# EPICS StreamDevice protocol: gemorcSup/devgemorc.proto
OutTerminator = CR;
InTerminator = CR;

getID {
	out "id";
	in "%#s";
}

initialise {
	out "in";
	in "OK";
}

re_zero_to_datum {
	out "da";
	in "OK";
}

stopNextInit {
	out "si";
	in "OK";
}

start {
	out "st";
	in "OK";
}

stop {
	out "sp";
	in "OK";
}

setWidth {
	out "ww%03d";
	in "OK";
	@init {out "rq"; in "%*16c%03d%*#s";}
}

setOffset {
	out "of%+04d";
	in "OK";
	@init {out "rq"; in "%*24c%04d%*#s";}
}

setSpeed {
	out "ds%03d";
	in "OK";
	@init {out "rq"; in "%*34c%02d%*#s";}
}

setAcc {
	out "ac%04d";
	in "OK";
	@init {out "rq"; in "%*41c%03d%*#s";}
}

getStatus {
    out "rq";
	# A:Oscillating[0:1], B:initialising[5:6], C:initialised_once[10:11], D:width[16:19], E:offset[24:28], F:speed[34:36], G:acceleration[41:44], H:cycles[46:51], I:backlash[61:64]
	in "%(\$1.A)01d%*4c%(\$1.B)01d%*4c%(\$1.C)01d%*5c%(\$1.D)03d%*6c%(\$1.E)+04d%*6c%(\$1.F)02d%*5c%(\$1.G)03d%*2c%(\$1.H)05d%*10c%(\$1.I)03d";
}
